TYPE ST_Machine_ServiceStatus :
STRUCT
	GC : ST_GC_ServiceStatus;
END_STRUCT
END_TYPE

(* stored: Version 1.1.0.1, ProductVersion 3.1.4026.18
   DUT ST_Machine_ServiceStatus: Id {42552cf1-31a3-48f9-b35d-49bb081e3583} *)
